FUNCTION_BLOCK EL6601
VAR
	{attribute addProperty Name "Info data"}
	_infoData : InfoDataAds;
END_VAR

END_FUNCTION_BLOCK

(* stored: Version 1.1.0.1, ProductVersion 3.1.4024.9
   POU EL6601: Id {d30ef104-5d01-04ac-1565-d0f451498cf9}, SpecialFunc None *)
